PROGRAM PRG_Thermocouple
VAR
	fTemp: REAL;
END_VAR

fTemp := GVL_Thermocouple.nTemp;

END_PROGRAM

(* stored: Version 1.1.0.1, ProductVersion 3.1.4024.12
   POU PRG_Thermocouple: Id {e6cc8783-084e-4bc3-b764-ac1c0275a869}, SpecialFunc None *)
